(* PLC project Unnamed, Unknown Unnamed 1 *)
(* stored: creationDateTime 2025-11-19T17:39:45, modificationDateTime 2025-11-19T18:11:09 *)

PROGRAM Task1
  VAR
    Start AT %IX0.1 : BOOL;
    Stop AT %IX0.0 : BOOL;
  END_VAR
  VAR
    Latch : BOOL;
  END_VAR
  VAR
    LED AT %QX0.0 : BOOL;
  END_VAR

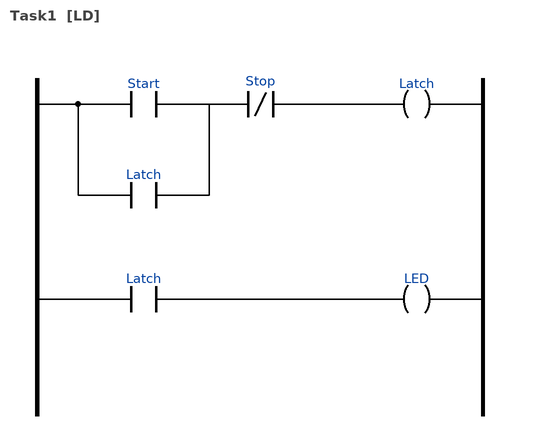
(* LD diagram, written out as Structured Text *)
Latch := (Start OR Latch) AND NOT Stop;
LED := Latch;
END_PROGRAM

CONFIGURATION Config0
  RESOURCE Res0 ON PLC
    TASK task0(INTERVAL := T#20ms, PRIORITY := 0);
    PROGRAM instance0 WITH task0 : Task1;
  END_RESOURCE
END_CONFIGURATION
